FUNCTION_BLOCK write_to_Buffer
VAR_INPUT
	m: REAL;
	startrecord : BOOL;
END_VAR
VAR_OUTPUT
	Datensatz : Datensatz;
	TimestampSYS: TIMESTRUCT;
END_VAR
VAR
	GetTime : NT_GetTime;
	GETTIMESTART : BOOL :=TRUE;
	Timestamp : T_Filetime;
	MyTimer: getsystemtime;
END_VAR

//100 values in array
	//GetTime(START := GETTIMESTART,TIMESTR => Timestamp);
	//Datensatz.Timestamp := SYSTEMTIME_TO_STRING(Timestamp);
	
	
	MyTimer();
	IF startrecord THEN
		Timestamp.dwLowDateTime:= MyTimer.timeLoDW;							
		Timestamp.dwHighDateTime := MyTimer.timeHiDW;
		TimestampSYS := FILETIME_TO_SYSTEMTIME(Timestamp);
		Datensatz.Timestamp := SYSTEMTIME_TO_STRING(TimestampSYS);
	END_IF
	Datensatz.temp := m;
	Datensatz.roomnum := 0.99999+m; 	
	Datensatz.signal3 := 20.99999+m;
	Datensatz.signal4 := 21.99999+m;
	Datensatz.signal5 := 22.99999+m;
	Datensatz.signal6 := 23.99999+m;
	Datensatz.signal7 := 24.99999+m;
	Datensatz.signal8 := 25.99999+m;

END_FUNCTION_BLOCK

(* stored: Version 1.1.0.1, ProductVersion 3.1.4024.3
   POU write_to_Buffer: Id {6ee574f5-f6d2-45c3-8dcf-06b67e67e4e2}, SpecialFunc None *)
